// LS Electric XG5000 project: 최종 plc 프레임_변경안2
// PLC LSPLC

PROGRAM 50_SerialComm (task: 스캔 프로그램)

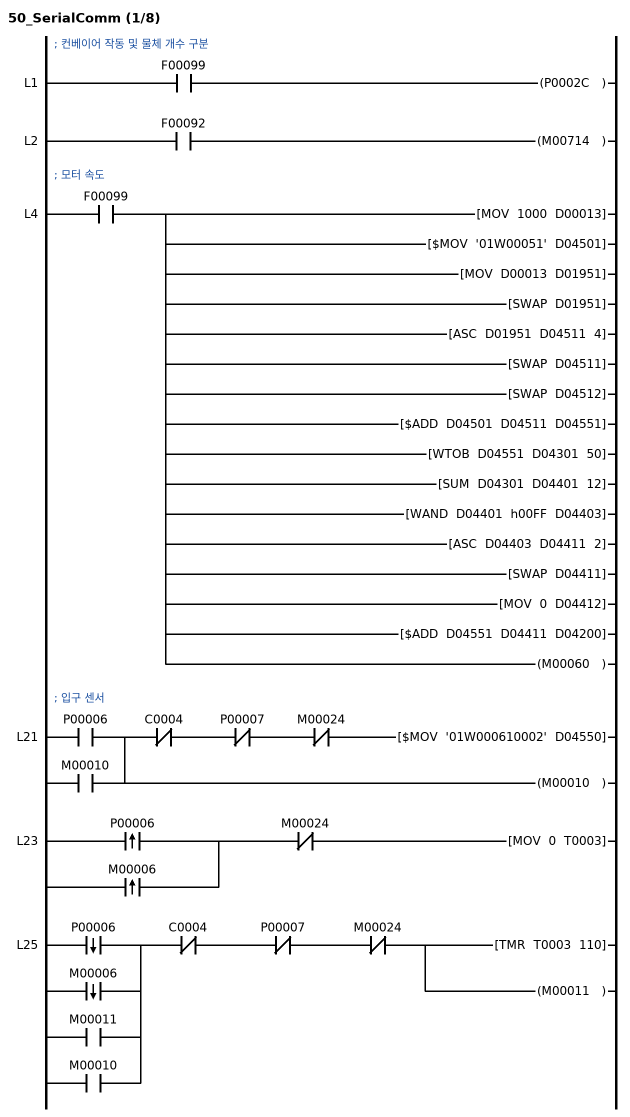
// 컨베이어 작동 및 물체 개수 구분
; L1
LOAD      F00099
OUT       P0002C
; L2
LOAD      F00092
OUT       M00714
// 모터 속도
; L4
LOAD      F00099
MOV       1000 D00013
$MOV      '01W00051' D04501
MOV       D00013 D01951
SWAP      D01951
ASC       D01951 D04511 4
SWAP      D04511
SWAP      D04512
$ADD      D04501 D04511 D04551
WTOB      D04551 D04301 50
SUM       D04301 D04401 12
WAND      D04401 h00FF D04403
ASC       D04403 D04411 2
SWAP      D04411
MOV       0 D04412
$ADD      D04551 D04411 D04200
OUT       M00060
// 입구 센서
; L21
LOAD      P00006
OR        M00010
MPUSH
AND NOT   C0004
AND NOT   P00007
AND NOT   M00024
$MOV      '01W000610002' D04550
MPOP
OUT       M00010
; L23
LOADP     P00006
ORP       M00006
AND NOT   M00024
MOV       0 T0003
; L25
LOADN     P00006
ORN       M00006
OR        M00011
OR        M00010
AND NOT   C0004
AND NOT   P00007
AND NOT   M00024
TMR       T0003 110
OUT       M00011

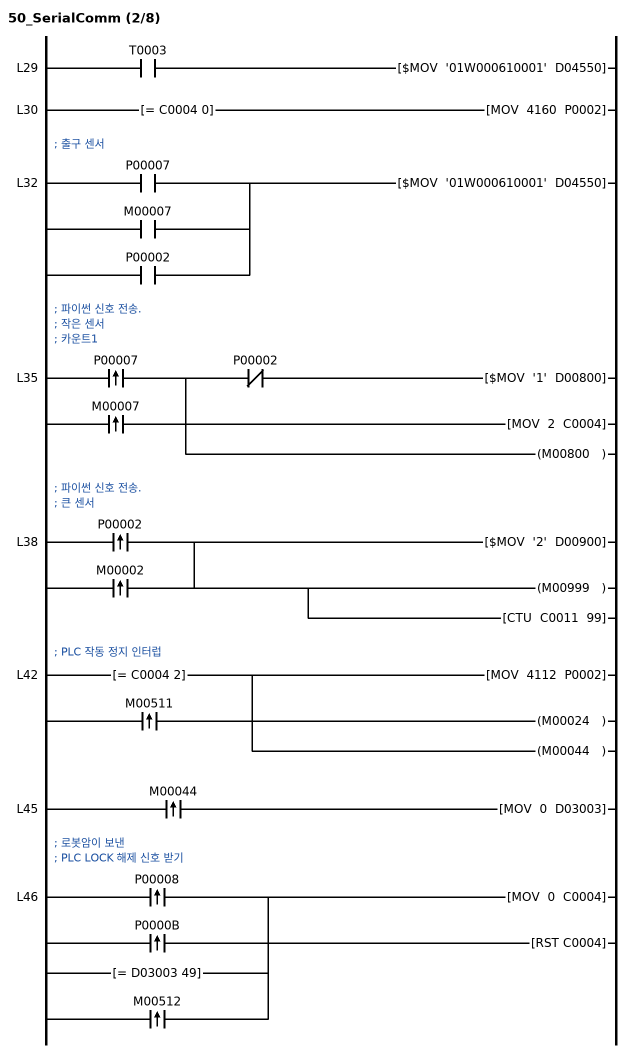
; L29
LOAD      T0003
$MOV      '01W000610001' D04550
; L30
LOAD=     C0004 0
MOV       4160 P0002
// 출구 센서
; L32
LOAD      P00007
OR        M00007
OR        P00002
$MOV      '01W000610001' D04550
; L35
LOADP     P00007
ORP       M00007
MPUSH
AND NOT   P00002
$MOV      '1' D00800
MPOP
MOV       2 C0004
OUT       M00800
// output comment: 파이썬 신호 전송. 작은 센서
// output comment: 카운트1
; L38
LOADP     P00002
ORP       M00002
$MOV      '2' D00900
OUT       M00999
CTU       C0011 99
// output comment: 파이썬 신호 전송. 큰 센서
; L42
LOAD=     C0004 2
ORP       M00511
MOV       4112 P0002
OUT       M00024
OUT       M00044
// output comment: PLC 작동 정지 인터럽
; L45
LOADP     M00044
MOV       0 D03003
; L46
LOADP     P00008
ORP       P0000B
OR=       D03003 49
ORP       M00512
MOV       0 C0004
RST       C0004
// output comment: 로봇암이 보낸 PLC LOCK 해제 신호 받기

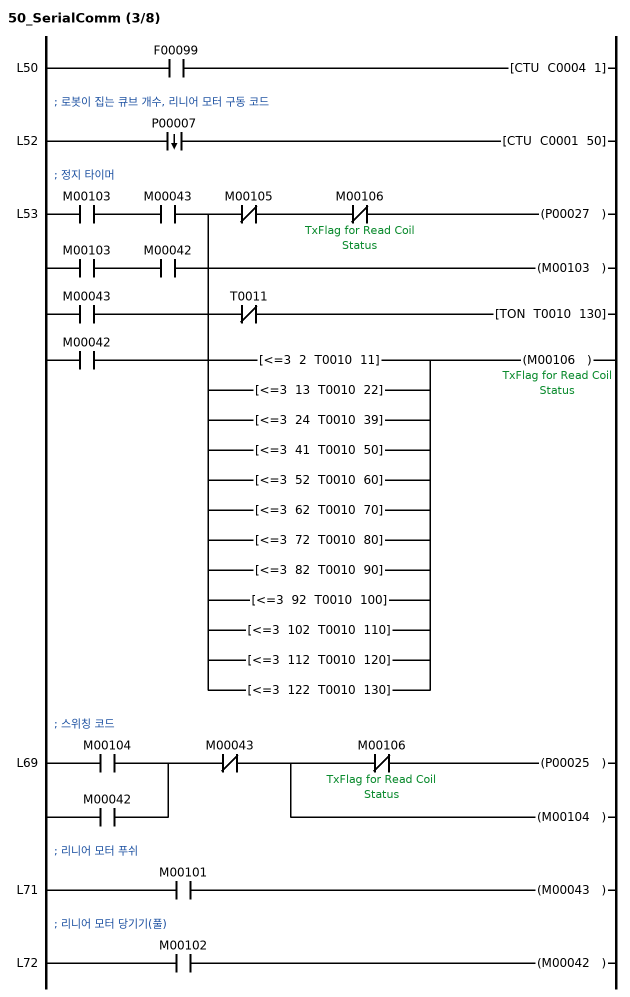
; L50
LOAD      F00099
CTU       C0004 1
// 로봇이 집는 큐브 개수, 리니어 모터 구동 코드
; L52
LOADN     P00007
CTU       C0001 50
; L53
LOAD      M00103
AND       M00043
LOAD      M00103
AND       M00042
OR LOAD
OR        M00043
OR        M00042
MPUSH
AND NOT   M00105
AND NOT   M00106	// TxFlag for Read Coil Status
OUT       P00027
MLOAD
OUT       M00103
AND NOT   T0011
TON       T0010 130
MPOP
LOAD<=3   2 T0010 11
OR<=3     13 T0010 22
OR<=3     24 T0010 39
OR<=3     41 T0010 50
OR<=3     52 T0010 60
OR<=3     62 T0010 70
OR<=3     72 T0010 80
OR<=3     82 T0010 90
OR<=3     92 T0010 100
OR<=3     102 T0010 110
OR<=3     112 T0010 120
OR<=3     122 T0010 130
AND LOAD
OUT       M00106	// TxFlag for Read Coil Status
// output comment: 정지 타이머
; L69
LOAD      M00104
OR        M00042
AND NOT   M00043
MPUSH
AND NOT   M00106	// TxFlag for Read Coil Status
OUT       P00025
MPOP
OUT       M00104
// output comment: 스위칭 코드
; L71
LOAD      M00101
OUT       M00043
// output comment: 리니어 모터 푸쉬
; L72
LOAD      M00102
OUT       M00042
// output comment: 리니어 모터 당기기(풀)

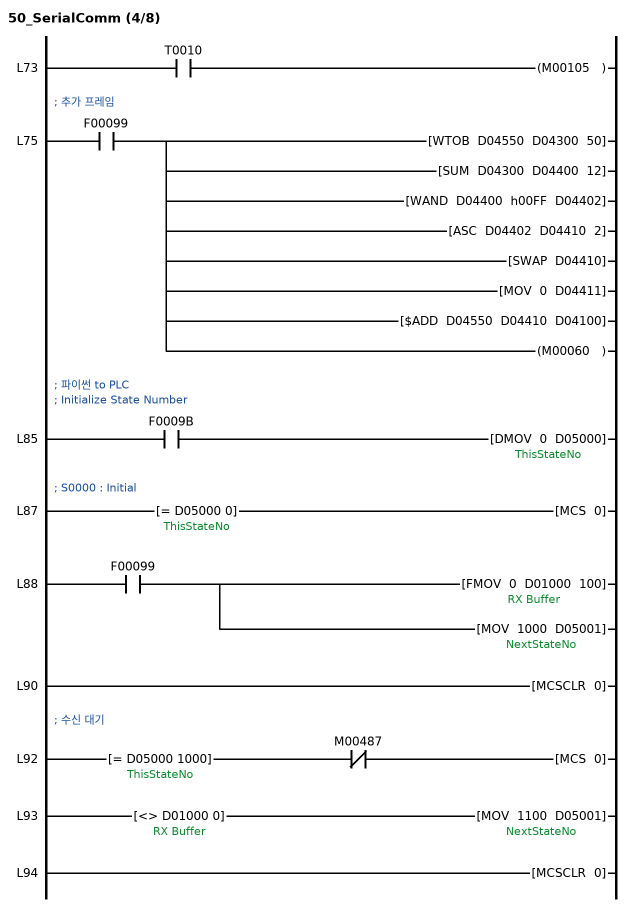
; L73
LOAD      T0010
OUT       M00105
// 추가 프레임
; L75
LOAD      F00099
WTOB      D04550 D04300 50
SUM       D04300 D04400 12
WAND      D04400 h00FF D04402
ASC       D04402 D04410 2
SWAP      D04410
MOV       0 D04411
$ADD      D04550 D04410 D04100
OUT       M00060
// 파이썬 to PLC
// Initialize State Number
; L85
LOAD      F0009B
DMOV      0 D05000	// ThisStateNo
// S0000 : Initial
; L87
LOAD=     D05000 0	// ThisStateNo
MCS       0
; L88
LOAD      F00099
FMOV      0 D01000 100	// RX Buffer
MOV       1000 D05001	// NextStateNo
; L90
MCSCLR    0
// 수신 대기
; L92
LOAD=     D05000 1000	// ThisStateNo
AND NOT   M00487
MCS       0
; L93
LOAD<>    D01000 0	// RX Buffer
MOV       1100 D05001	// NextStateNo
; L94
MCSCLR    0

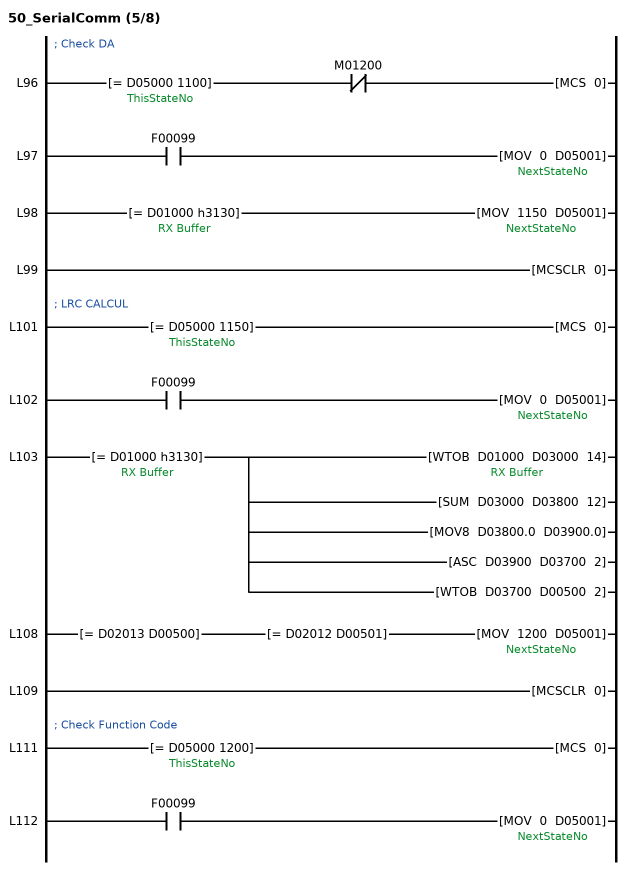
// Check DA
; L96
LOAD=     D05000 1100	// ThisStateNo
AND NOT   M01200
MCS       0
; L97
LOAD      F00099
MOV       0 D05001	// NextStateNo
; L98
LOAD=     D01000 h3130	// RX Buffer
MOV       1150 D05001	// NextStateNo
; L99
MCSCLR    0
// LRC CALCUL
; L101
LOAD=     D05000 1150	// ThisStateNo
MCS       0
; L102
LOAD      F00099
MOV       0 D05001	// NextStateNo
; L103
LOAD=     D01000 h3130	// RX Buffer
WTOB      D01000 D03000 14	// RX Buffer
SUM       D03000 D03800 12
MOV8      D03800.0 D03900.0
ASC       D03900 D03700 2
WTOB      D03700 D00500 2
; L108
LOAD=     D02013 D00500
AND=      D02012 D00501
MOV       1200 D05001	// NextStateNo
; L109
MCSCLR    0
// Check Function Code
; L111
LOAD=     D05000 1200	// ThisStateNo
MCS       0
; L112
LOAD      F00099
MOV       0 D05001	// NextStateNo

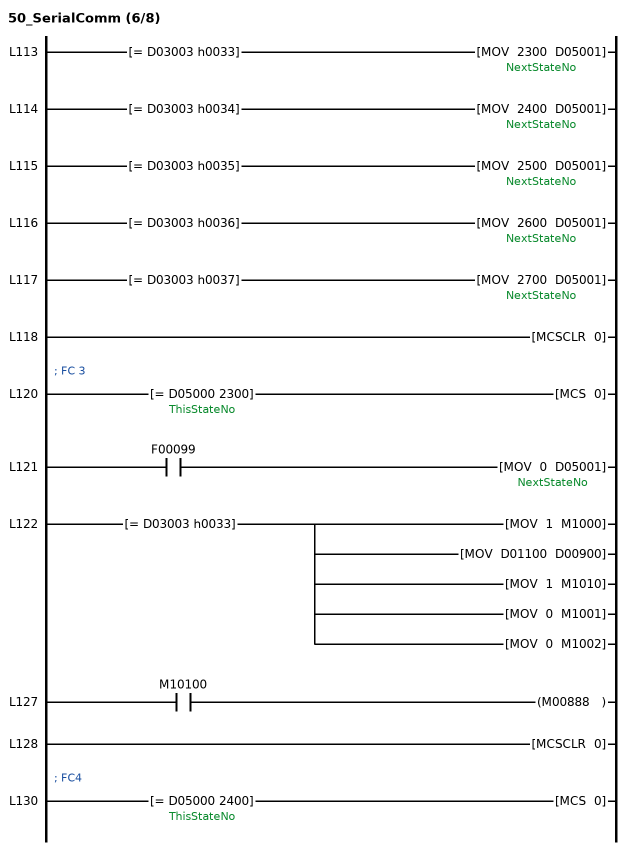
; L113
LOAD=     D03003 h0033
MOV       2300 D05001	// NextStateNo
; L114
LOAD=     D03003 h0034
MOV       2400 D05001	// NextStateNo
; L115
LOAD=     D03003 h0035
MOV       2500 D05001	// NextStateNo
; L116
LOAD=     D03003 h0036
MOV       2600 D05001	// NextStateNo
; L117
LOAD=     D03003 h0037
MOV       2700 D05001	// NextStateNo
; L118
MCSCLR    0
// FC 3
; L120
LOAD=     D05000 2300	// ThisStateNo
MCS       0
; L121
LOAD      F00099
MOV       0 D05001	// NextStateNo
; L122
LOAD=     D03003 h0033
MOV       1 M1000
MOV       D01100 D00900
MOV       1 M1010
MOV       0 M1001
MOV       0 M1002
; L127
LOAD      M10100
OUT       M00888
; L128
MCSCLR    0
// FC4
; L130
LOAD=     D05000 2400	// ThisStateNo
MCS       0

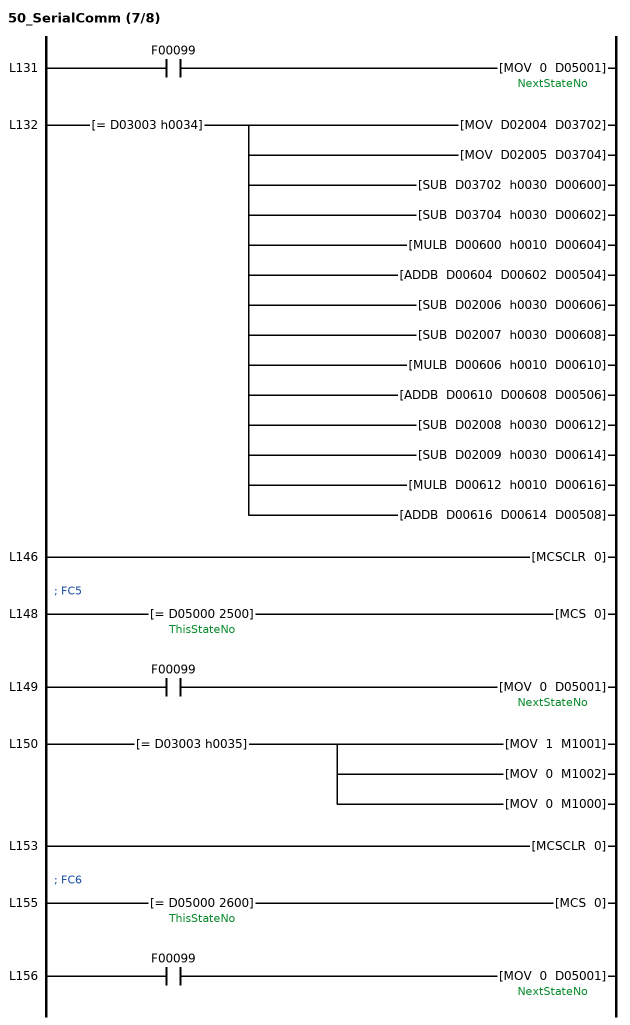
; L131
LOAD      F00099
MOV       0 D05001	// NextStateNo
; L132
LOAD=     D03003 h0034
MOV       D02004 D03702
MOV       D02005 D03704
SUB       D03702 h0030 D00600
SUB       D03704 h0030 D00602
MULB      D00600 h0010 D00604
ADDB      D00604 D00602 D00504
SUB       D02006 h0030 D00606
SUB       D02007 h0030 D00608
MULB      D00606 h0010 D00610
ADDB      D00610 D00608 D00506
SUB       D02008 h0030 D00612
SUB       D02009 h0030 D00614
MULB      D00612 h0010 D00616
ADDB      D00616 D00614 D00508
; L146
MCSCLR    0
// FC5
; L148
LOAD=     D05000 2500	// ThisStateNo
MCS       0
; L149
LOAD      F00099
MOV       0 D05001	// NextStateNo
; L150
LOAD=     D03003 h0035
MOV       1 M1001
MOV       0 M1002
MOV       0 M1000
; L153
MCSCLR    0
// FC6
; L155
LOAD=     D05000 2600	// ThisStateNo
MCS       0
; L156
LOAD      F00099
MOV       0 D05001	// NextStateNo

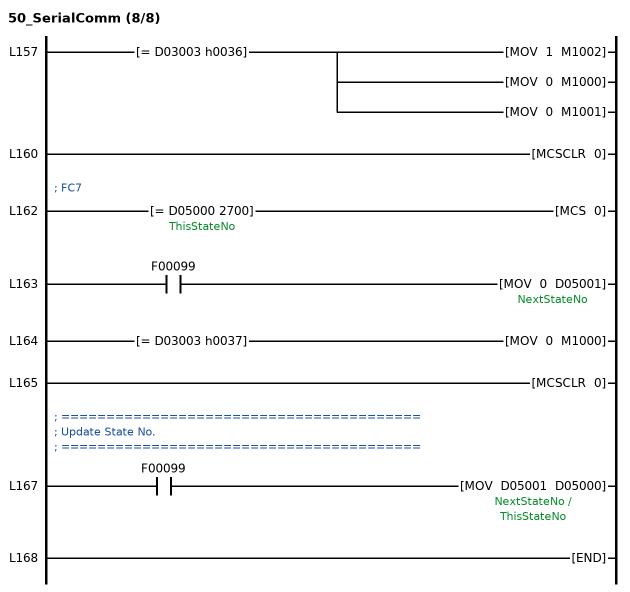
; L157
LOAD=     D03003 h0036
MOV       1 M1002
MOV       0 M1000
MOV       0 M1001
; L160
MCSCLR    0
// FC7
; L162
LOAD=     D05000 2700	// ThisStateNo
MCS       0
; L163
LOAD      F00099
MOV       0 D05001	// NextStateNo
; L164
LOAD=     D03003 h0037
MOV       0 M1000
; L165
MCSCLR    0
// ========================================
// Update State No.
// ========================================
; L167
LOAD      F00099
MOV       D05001 D05000	// NextStateNo / ThisStateNo
; L168
END

PROGRAM 60_TX_Flag (task: 스캔 프로그램)

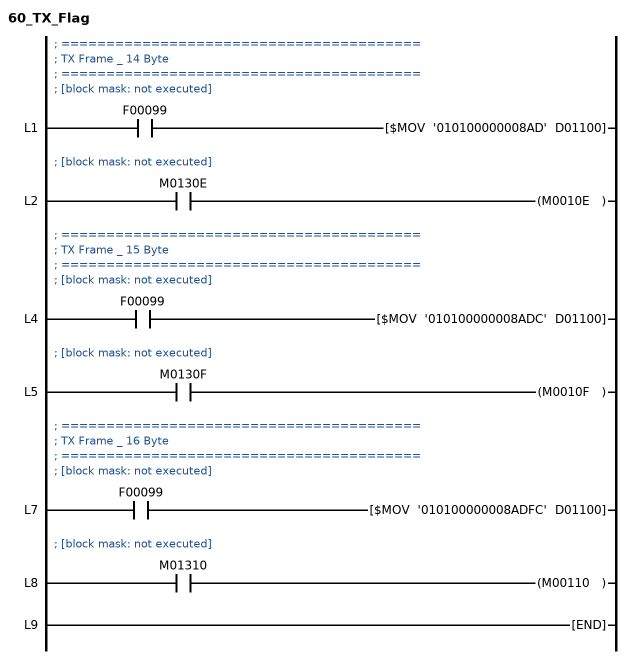
// ========================================
// TX Frame _ 14 Byte
// ========================================
; L1 (block mask: not executed)
LOAD      F00099
$MOV      '010100000008AD' D01100
; L2 (block mask: not executed)
LOAD      M0130E
OUT       M0010E
// ========================================
// TX Frame _ 15 Byte
// ========================================
; L4 (block mask: not executed)
LOAD      F00099
$MOV      '010100000008ADC' D01100
; L5 (block mask: not executed)
LOAD      M0130F
OUT       M0010F
// ========================================
// TX Frame _ 16 Byte
// ========================================
; L7 (block mask: not executed)
LOAD      F00099
$MOV      '010100000008ADFC' D01100
; L8 (block mask: not executed)
LOAD      M01310
OUT       M00110
; L9
END

PROGRAM convey (task: 스캔 프로그램)

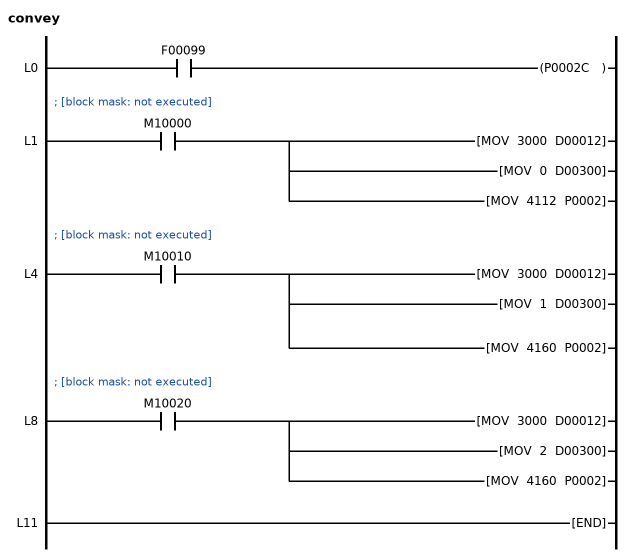
; L0
LOAD      F00099
OUT       P0002C
; L1 (block mask: not executed)
LOAD      M10000
MOV       3000 D00012
MOV       0 D00300
MOV       4112 P0002
; L4 (block mask: not executed)
LOAD      M10010
MOV       3000 D00012
MOV       1 D00300
MOV       4160 P0002
; L8 (block mask: not executed)
LOAD      M10020
MOV       3000 D00012
MOV       2 D00300
MOV       4160 P0002
; L11
END

PROGRAM tp_inter (task: 스캔 프로그램)

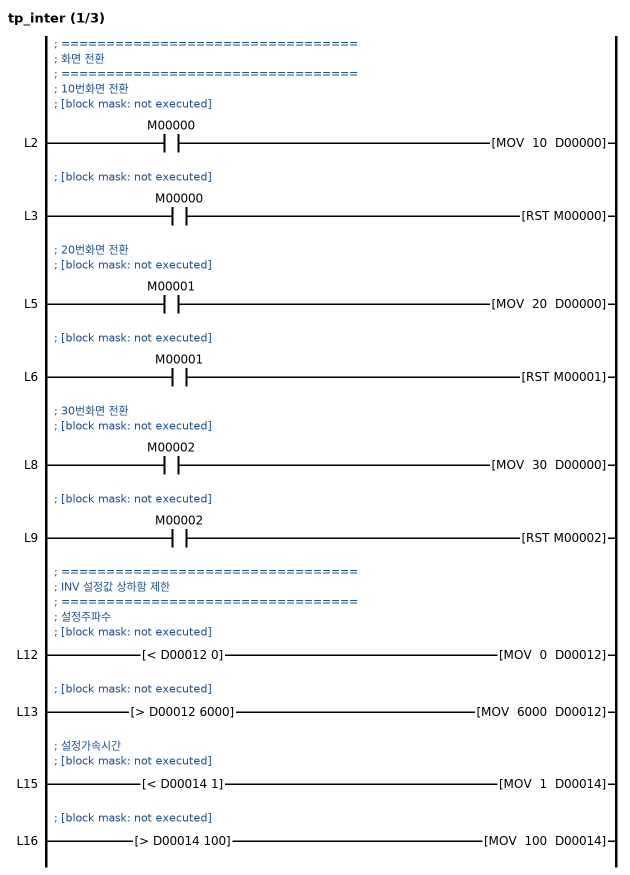
// =================================
//    화면 전환
// =================================
// 10번화면 전환
; L2 (block mask: not executed)
LOAD      M00000
MOV       10 D00000
; L3 (block mask: not executed)
LOAD      M00000
RST       M00000
// 20번화면 전환
; L5 (block mask: not executed)
LOAD      M00001
MOV       20 D00000
; L6 (block mask: not executed)
LOAD      M00001
RST       M00001
// 30번화면 전환
; L8 (block mask: not executed)
LOAD      M00002
MOV       30 D00000
; L9 (block mask: not executed)
LOAD      M00002
RST       M00002
// =================================
//    INV 설정값 상하함 제한
// =================================
// 설정주파수
; L12 (block mask: not executed)
LOAD<     D00012 0
MOV       0 D00012
; L13 (block mask: not executed)
LOAD>     D00012 6000
MOV       6000 D00012
// 설정가속시간
; L15 (block mask: not executed)
LOAD<     D00014 1
MOV       1 D00014
; L16 (block mask: not executed)
LOAD>     D00014 100
MOV       100 D00014

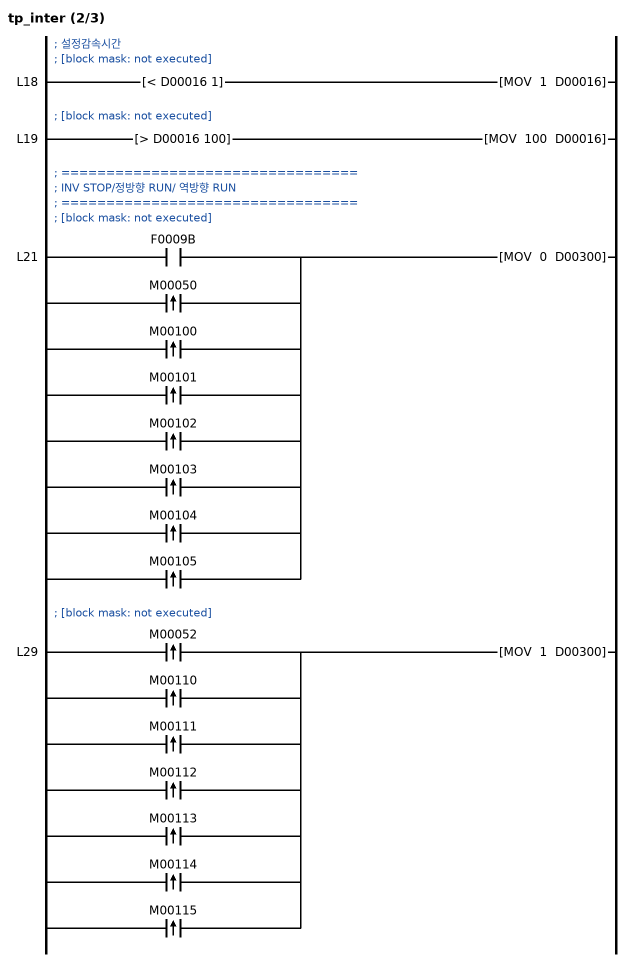
// 설정감속시간
; L18 (block mask: not executed)
LOAD<     D00016 1
MOV       1 D00016
; L19 (block mask: not executed)
LOAD>     D00016 100
MOV       100 D00016
// =================================
//    INV STOP/정방향 RUN/ 역방향 RUN
// =================================
; L21 (block mask: not executed)
LOAD      F0009B
ORP       M00050
ORP       M00100
ORP       M00101
ORP       M00102
ORP       M00103
ORP       M00104
ORP       M00105
MOV       0 D00300
; L29 (block mask: not executed)
LOADP     M00052
ORP       M00110
ORP       M00111
ORP       M00112
ORP       M00113
ORP       M00114
ORP       M00115
MOV       1 D00300

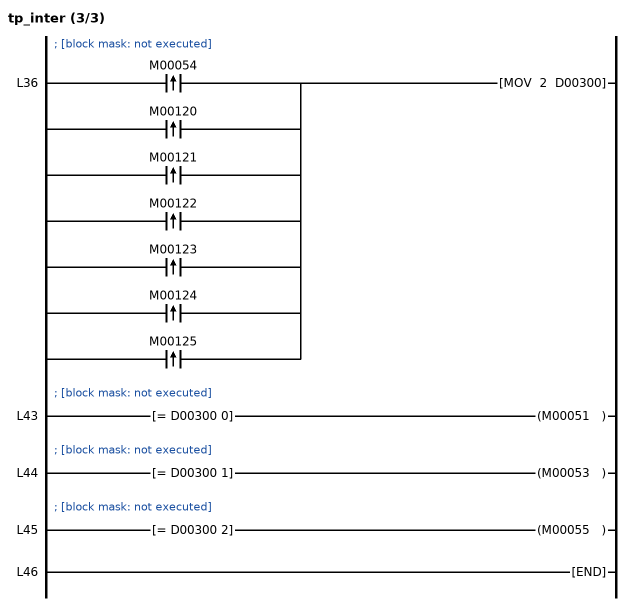
; L36 (block mask: not executed)
LOADP     M00054
ORP       M00120
ORP       M00121
ORP       M00122
ORP       M00123
ORP       M00124
ORP       M00125
MOV       2 D00300
; L43 (block mask: not executed)
LOAD=     D00300 0
OUT       M00051
; L44 (block mask: not executed)
LOAD=     D00300 1
OUT       M00053
; L45 (block mask: not executed)
LOAD=     D00300 2
OUT       M00055
; L46
END

PROGRAM inv (task: 스캔 프로그램)

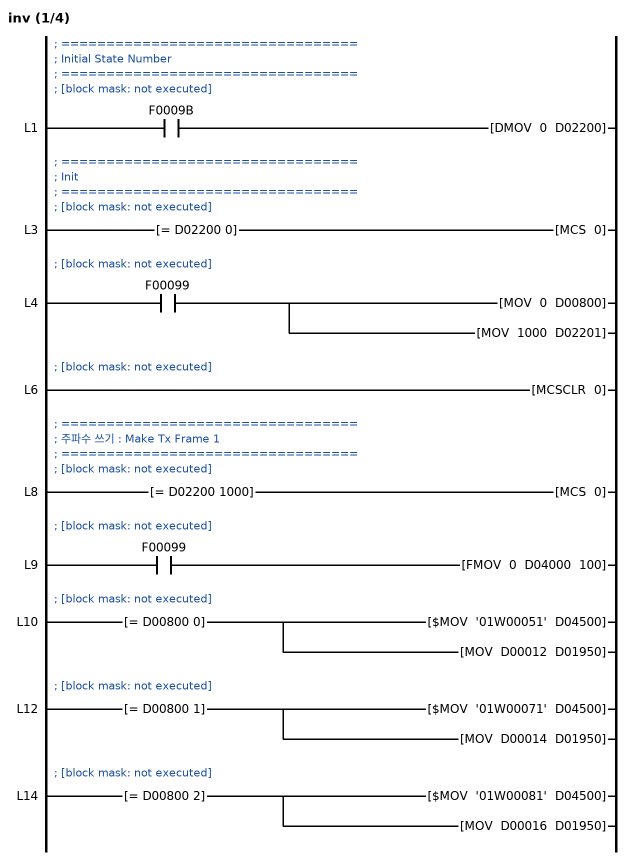
// =================================
//    Initial State Number
// =================================
; L1 (block mask: not executed)
LOAD      F0009B
DMOV      0 D02200
// =================================
//    Init
// =================================
; L3 (block mask: not executed)
LOAD=     D02200 0
MCS       0
; L4 (block mask: not executed)
LOAD      F00099
MOV       0 D00800
MOV       1000 D02201
; L6 (block mask: not executed)
MCSCLR    0
// =================================
//    주파수 쓰기 : Make Tx Frame 1
// =================================
; L8 (block mask: not executed)
LOAD=     D02200 1000
MCS       0
; L9 (block mask: not executed)
LOAD      F00099
FMOV      0 D04000 100
; L10 (block mask: not executed)
LOAD=     D00800 0
$MOV      '01W00051' D04500
MOV       D00012 D01950
; L12 (block mask: not executed)
LOAD=     D00800 1
$MOV      '01W00071' D04500
MOV       D00014 D01950
; L14 (block mask: not executed)
LOAD=     D00800 2
$MOV      '01W00081' D04500
MOV       D00016 D01950

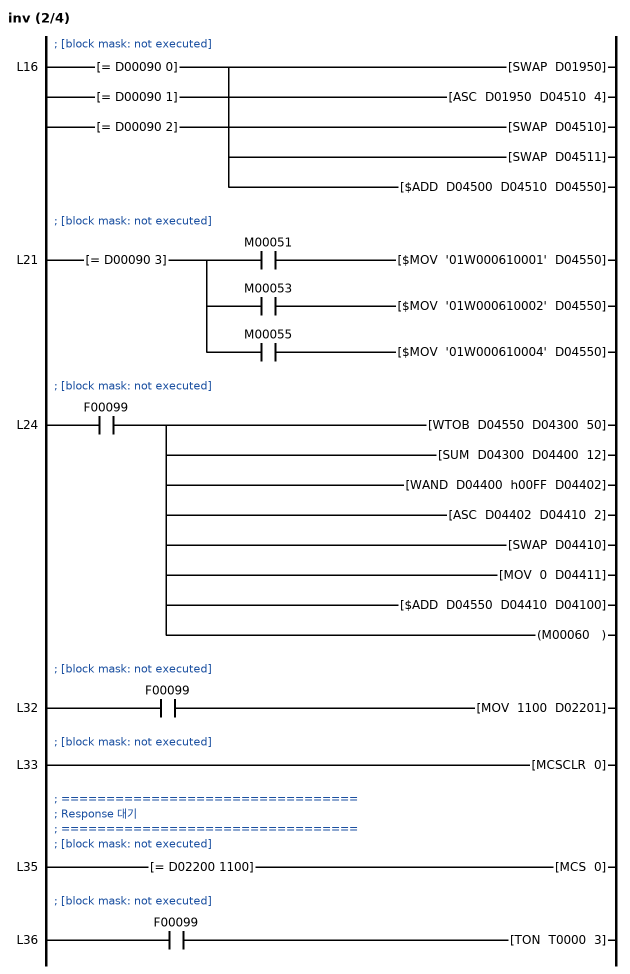
; L16 (block mask: not executed)
LOAD=     D00090 0
OR=       D00090 1
OR=       D00090 2
SWAP      D01950
ASC       D01950 D04510 4
SWAP      D04510
SWAP      D04511
$ADD      D04500 D04510 D04550
; L21 (block mask: not executed)
LOAD=     D00090 3
MPUSH
AND       M00051
$MOV      '01W000610001' D04550
MLOAD
AND       M00053
$MOV      '01W000610002' D04550
MPOP
AND       M00055
$MOV      '01W000610004' D04550
; L24 (block mask: not executed)
LOAD      F00099
WTOB      D04550 D04300 50
SUM       D04300 D04400 12
WAND      D04400 h00FF D04402
ASC       D04402 D04410 2
SWAP      D04410
MOV       0 D04411
$ADD      D04550 D04410 D04100
OUT       M00060
; L32 (block mask: not executed)
LOAD      F00099
MOV       1100 D02201
; L33 (block mask: not executed)
MCSCLR    0
// =================================
//    Response 대기
// =================================
; L35 (block mask: not executed)
LOAD=     D02200 1100
MCS       0
; L36 (block mask: not executed)
LOAD      F00099
TON       T0000 3

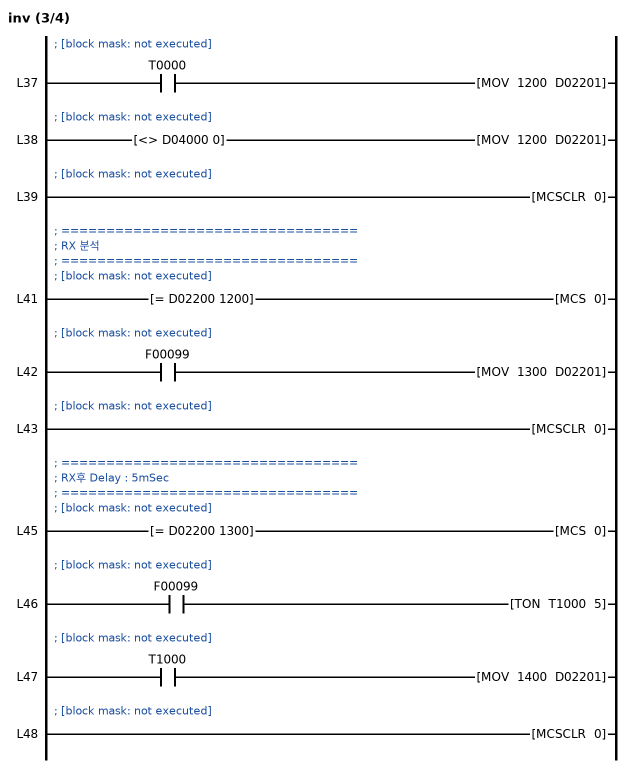
; L37 (block mask: not executed)
LOAD      T0000
MOV       1200 D02201
; L38 (block mask: not executed)
LOAD<>    D04000 0
MOV       1200 D02201
; L39 (block mask: not executed)
MCSCLR    0
// =================================
//    RX 분석
// =================================
; L41 (block mask: not executed)
LOAD=     D02200 1200
MCS       0
; L42 (block mask: not executed)
LOAD      F00099
MOV       1300 D02201
; L43 (block mask: not executed)
MCSCLR    0
// =================================
//    RX후 Delay : 5mSec
// =================================
; L45 (block mask: not executed)
LOAD=     D02200 1300
MCS       0
; L46 (block mask: not executed)
LOAD      F00099
TON       T1000 5
; L47 (block mask: not executed)
LOAD      T1000
MOV       1400 D02201
; L48 (block mask: not executed)
MCSCLR    0

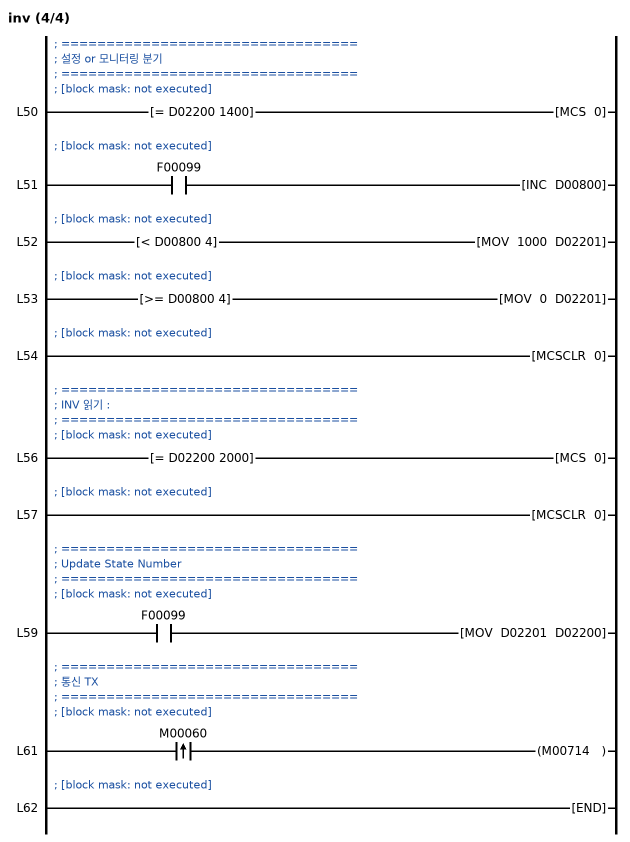
// =================================
//    설정 or 모니터링 분기
// =================================
; L50 (block mask: not executed)
LOAD=     D02200 1400
MCS       0
; L51 (block mask: not executed)
LOAD      F00099
INC       D00800
; L52 (block mask: not executed)
LOAD<     D00800 4
MOV       1000 D02201
; L53 (block mask: not executed)
LOAD>=    D00800 4
MOV       0 D02201
; L54 (block mask: not executed)
MCSCLR    0
// =================================
//    INV 읽기 :
// =================================
; L56 (block mask: not executed)
LOAD=     D02200 2000
MCS       0
; L57 (block mask: not executed)
MCSCLR    0
// =================================
//    Update State Number
// =================================
; L59 (block mask: not executed)
LOAD      F00099
MOV       D02201 D02200
// =================================
//    통신 TX
// =================================
; L61 (block mask: not executed)
LOADP     M00060
OUT       M00714
; L62 (block mask: not executed)
END

VARIABLES AND COMMENTS (devices not used above)
D02001	WORD	RX Function Code
D03500	WORD	연산 CRC
D03562	WORD	수신 CRC
D03560	WORD	CRC 연산할 Byte 수